{attribute 'GeneratedUsingTerminal: EL6201-0000-0017'}
{attribute addProperty BoxType "EL6201-0000-0017"}
{attribute addProperty Id "Auto_Programming_EnableAT %Q*BOOL1Go_Offline_ModeAT %Q*BOOL1Data_Exchange_ActiveAT %Q*BOOL1Go_Protected_ModeAT %Q*BOOL1Go_Configuration_ModeAT %Q*BOOL1"}
{attribute addProperty CRC "4099653163"}
{attribute addProperty Size "5"}
TYPE ASI_Control_F45BBE2B :
STRUCT
	{attribute addProperty Name "Auto_Programming_Enable"}
	Auto_Programming_Enable AT %Q* : BOOL;
	{attribute addProperty Name "Go_Offline_Mode"}
	Go_Offline_Mode AT %Q* : BOOL;
	{attribute addProperty Name "Data_Exchange_Active"}
	Data_Exchange_Active AT %Q* : BOOL;
	{attribute addProperty Name "Go_Protected_Mode"}
	Go_Protected_Mode AT %Q* : BOOL;
	{attribute addProperty Name "Go_Configuration_Mode"}
	Go_Configuration_Mode AT %Q* : BOOL;
END_STRUCT
END_TYPE

(* stored: Version 1.2.0.0, ProductVersion 3.1.4024.9
   DUT ASI_Control_F45BBE2B: Id {98873546-9b2f-4c41-b08c-29fc97efc99f} *)
